FUNCTION_BLOCK {BlockName} (* {Description} *)
  (* Standard: 61499-2 *)
  (* Version 0.0, {MM/DD/YYYY}, {Author}, {YourOrg}, Initial version *)
  PACKAGE {YourNamespace};
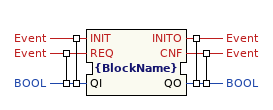
  EVENT_INPUT
    INIT WITH QI; (* Initialization Request *)
    REQ WITH QI; (* Normal Execution Request *)
  END_EVENT
  EVENT_OUTPUT
    INITO WITH QO; (* Initialization Confirm *)
    CNF WITH QO; (* Execution Confirmation *)
  END_EVENT
  VAR_INPUT
    QI : BOOL; (* Input event qualifier *)
  END_VAR
  VAR_OUTPUT
    QO : BOOL; (* Output event qualifier *)
  END_VAR
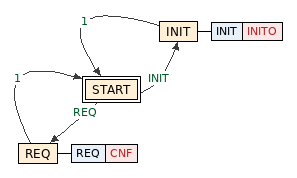
  EC_STATES
    START; (* Initial State *)
    INIT : INIT -> INITO; (* Initialization *)
    REQ : REQ -> CNF; (* Normal execution *)
  END_STATES
  EC_TRANSITIONS
    START TO INIT := INIT;
    INIT TO START := 1;
    START TO REQ := REQ;
    REQ TO START := 1;
  END_TRANSITIONS
  ALGORITHM INIT IN ST: (* Initialization algorithm *)
{INIT_ALGORITHM_CODE}
  END_ALGORITHM
  ALGORITHM REQ IN ST: (* Normally executed algorithm *)
{REQ_ALGORITHM_CODE}
  END_ALGORITHM
END_FUNCTION_BLOCK
